# EPICS autosave request: iocBoot/ioc13idd/auto_positions.req
file "CARS_88_motor_positions.req", P=$(P)
